INTERFACE Value EXTENDS ValueRead

METHOD Set
VAR_INPUT
END_VAR
END_METHOD

END_INTERFACE

(* stored: Version 1.1.0.1, ProductVersion 3.1.4024.15
   Itf Value: Id {005347b3-e21f-4935-9d8b-47c49c306fc1}
   Method Set: Id {50cd76fe-4b86-41a4-9aa5-f7103323bb6a} *)
